FUNCTION_BLOCK TrojanUV3000 (* Composite Function Block Type *)
  (* Standard: 61499-2 *)
  (* Version 0.0, 03/03/2026, template *)
  PACKAGE Hidryco.HidrycoLib;
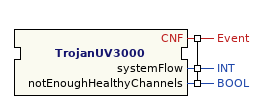
  EVENT_OUTPUT
    CNF WITH systemFlow, notEnoughHealthyChannels;
  END_EVENT
  VAR_OUTPUT
    systemFlow : INT;
    notEnoughHealthyChannels : BOOL;
  END_VAR
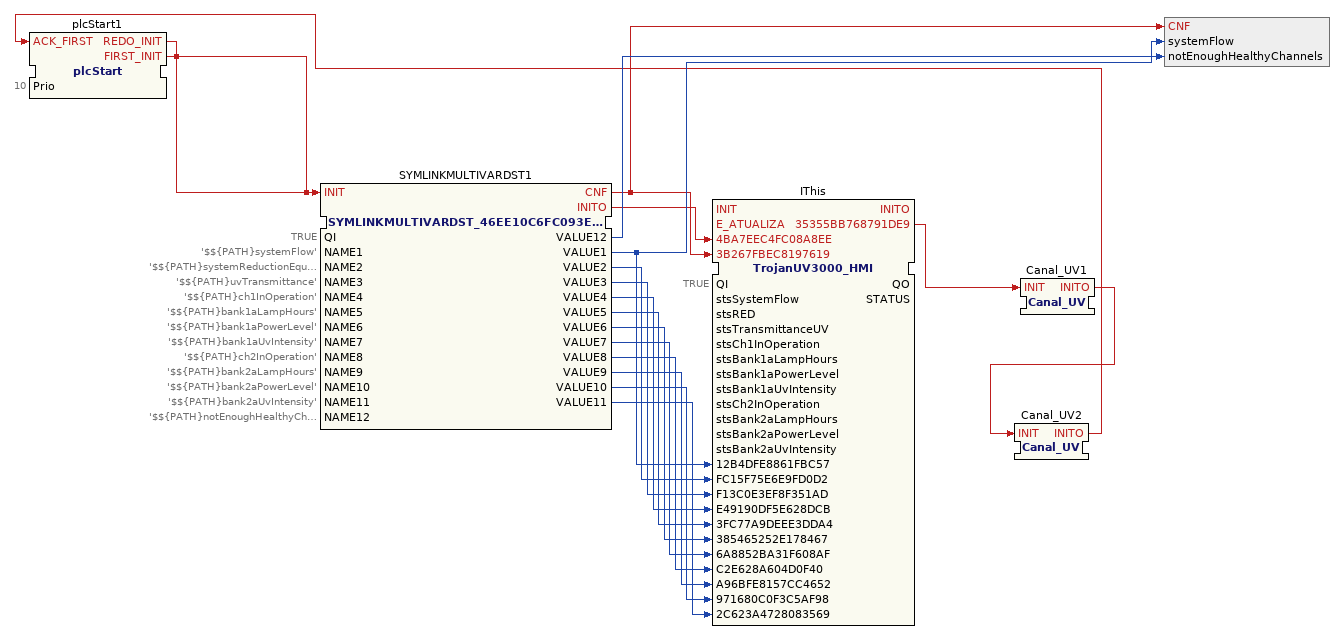
  FBS
    Canal_UV1 : Canal_UV;
    Canal_UV2 : Canal_UV;
    SYMLINKMULTIVARDST1 : SYMLINKMULTIVARDST_46EE10C6FC093EFB(QI := TRUE, NAME1 := '$${PATH}systemFlow' {SET_ATTRIBUTE(Configuration.Parameter.Style, Width=200)}, NAME2 := '$${PATH}systemReductionEquivalentDose' {SET_ATTRIBUTE(Configuration.Parameter.Style, Width=200)}, NAME3 := '$${PATH}uvTransmittance' {SET_ATTRIBUTE(Configuration.Parameter.Style, Width=200)}, NAME4 := '$${PATH}ch1InOperation' {SET_ATTRIBUTE(Configuration.Parameter.Style, Width=200)}, NAME5 := '$${PATH}bank1aLampHours' {SET_ATTRIBUTE(Configuration.Parameter.Style, Width=200)}, NAME6 := '$${PATH}bank1aPowerLevel' {SET_ATTRIBUTE(Configuration.Parameter.Style, Width=200)}, NAME7 := '$${PATH}bank1aUvIntensity' {SET_ATTRIBUTE(Configuration.Parameter.Style, Width=200)}, NAME8 := '$${PATH}ch2InOperation' {SET_ATTRIBUTE(Configuration.Parameter.Style, Width=200)}, NAME9 := '$${PATH}bank2aLampHours' {SET_ATTRIBUTE(Configuration.Parameter.Style, Width=200)}, NAME10 := '$${PATH}bank2aPowerLevel' {SET_ATTRIBUTE(Configuration.Parameter.Style, Width=200)}, NAME11 := '$${PATH}bank2aUvIntensity' {SET_ATTRIBUTE(Configuration.Parameter.Style, Width=200)}, NAME12 := '$${PATH}notEnoughHealthyChannels'); {SET_ATTRIBUTE(Configuration.GenericFBType.InterfaceParams, Runtime.System#I:=13;VALUE${I$}:INT,INT,INT,BOOL,INT,INT,INT,BOOL,INT,INT,INT,BOOL,INT)}
    plcStart1 : plcStart(Prio := 10);
    IThis : TrojanUV3000_HMI(QI := TRUE);
  END_FBS
  EVENT_CONNECTIONS
    Canal_UV2.INITO TO plcStart1.ACK_FIRST;
    Canal_UV1.INITO TO Canal_UV2.INIT;
    plcStart1.REDO_INIT TO SYMLINKMULTIVARDST1.INIT;
    plcStart1.FIRST_INIT TO SYMLINKMULTIVARDST1.INIT;
    SYMLINKMULTIVARDST1.CNF TO CNF;
    SYMLINKMULTIVARDST1.INITO TO IThis.4BA7EEC4FC08A8EE;
    SYMLINKMULTIVARDST1.CNF TO IThis.3B267FBEC8197619;
    IThis.35355BB768791DE9 TO Canal_UV1.INIT;
  END_CONNECTIONS
  DATA_CONNECTIONS
    SYMLINKMULTIVARDST1.VALUE12 TO notEnoughHealthyChannels;
    SYMLINKMULTIVARDST1.VALUE1 TO systemFlow;
    SYMLINKMULTIVARDST1.VALUE1 TO IThis.12B4DFE8861FBC57;
    SYMLINKMULTIVARDST1.VALUE2 TO IThis.FC15F75E6E9FD0D2;
    SYMLINKMULTIVARDST1.VALUE3 TO IThis.F13C0E3EF8F351AD;
    SYMLINKMULTIVARDST1.VALUE4 TO IThis.E49190DF5E628DCB;
    SYMLINKMULTIVARDST1.VALUE5 TO IThis.3FC77A9DEEE3DDA4;
    SYMLINKMULTIVARDST1.VALUE6 TO IThis.385465252E178467;
    SYMLINKMULTIVARDST1.VALUE7 TO IThis.6A8852BA31F608AF;
    SYMLINKMULTIVARDST1.VALUE8 TO IThis.C2E628A604D0F40;
    SYMLINKMULTIVARDST1.VALUE9 TO IThis.A96BFE8157CC4652;
    SYMLINKMULTIVARDST1.VALUE10 TO IThis.971680C0F3C5AF98;
    SYMLINKMULTIVARDST1.VALUE11 TO IThis.2C623A4728083569;
  END_CONNECTIONS
END_FUNCTION_BLOCK
